Universal Robots PolyScope program: Group21Lab1Task3.urp

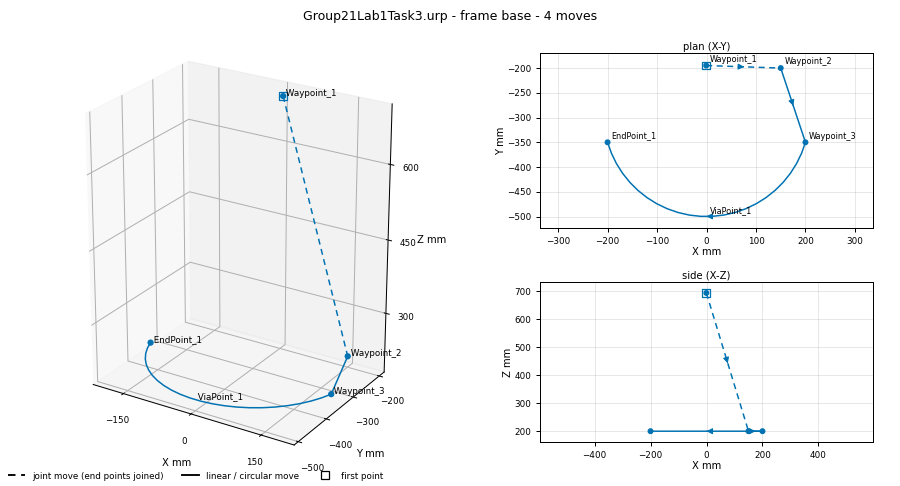
[picture p0: tool path of Group21Lab1Task3.urp in frame base, 4 of 5 moves have a stored position in this frame; points joined in program order, loops and branches not executed]
Program group21p3 (createdIn=3.5.0.10584 lastSavedIn=3.5.0.10584 directory=/programs/usbdisk installation=default robotSerialNumber=2017332505)
Calibrated DH parameters: a=[0, -0.24355, -0.210285, 0.000007, -0.000026, 0]; d=[0.151972, 1.341373, 3.010199, -4.239311, 0.085317, 0.082321]; alpha=[1.570715, -0.004846, 0.008121, 1.57079, -1.571065, 0]; deltaTheta=[0.000017, -0.02667, 0.193133, -0.166555, -0.000046, 0.000042]
Robot Program (runOnlyOnce=false motionType=MoveJ speed=1.047198 acceleration=1.396263 useActiveTCP=false)
  MoveJ speed 60 deg/s, acceleration 80 deg/s^2 (useActiveTCP=false)
    Waypoint Waypoint_1: TCP in base x=-0.573 y=-194.849 z=693.865 mm, rx=0 ry=-0.0016 rz=-0.0016 rad; joints [0, -90, 0, -90, 0, 0] deg
    Waypoint Waypoint_2: TCP in base x=150.006 y=-200.003 z=200.001 mm, rx=1.5699 ry=0 rz=0 rad; joints [-26.792, -79.435, -131.611, -59.037, 90.488, 63.559] deg
  MoveP speed 250 mm/s, acceleration 1200 mm/s^2 (blendRadius=0.025 useActiveTCP=false) feature=Base
    Waypoint Waypoint_3: TCP in base x=199.976 y=-350.024 z=199.996 mm, rx=1.57 ry=0 rz=-0.0002 rad; joints [-44.295, -116.253, -88.317, -65.514, 90.293, 45.981] deg
    CircleMove (OrientationMode=FIXED)
      Waypoint ViaPoint_1: TCP in base x=-0.029 y=-500.001 z=199.958 mm, rx=1.5701 ry=0.0001 rz=-0.0004 rad; joints [-77.105, -141.204, -44.908, -83.943, 90.162, 12.949] deg; flange x=0 y=-500 z=200 mm, rx=0.0023 ry=-3.1398 rz=-0.0015 rad
      Waypoint EndPoint_1: TCP in base x=-199.981 y=-349.988 z=199.969 mm, rx=1.5702 ry=0.0001 rz=-0.0003 rad; joints [-103.767, -116.233, -88.382, -65.391, 90.21, -13.483] deg
